PROGRAM ITMotion
VAR
	odometrie 			:FB_Motion_Odometrie;
END_VAR
VAR_INPUT
	IbPower				:BOOL;
	IbStop				:BOOL;
	IbPause				:BOOL;
	IbReset				:BOOL;
END_VAR
VAR_OUTPUT
	QbMoteurOn		:BOOL;
	QbMouvementTermine 	:BOOL;
END_VAR
VAR // added by the converter: edge detectors and wires of the graphical bodies
    _w1, _w2, _w3, _w4 : BOOL;
END_VAR

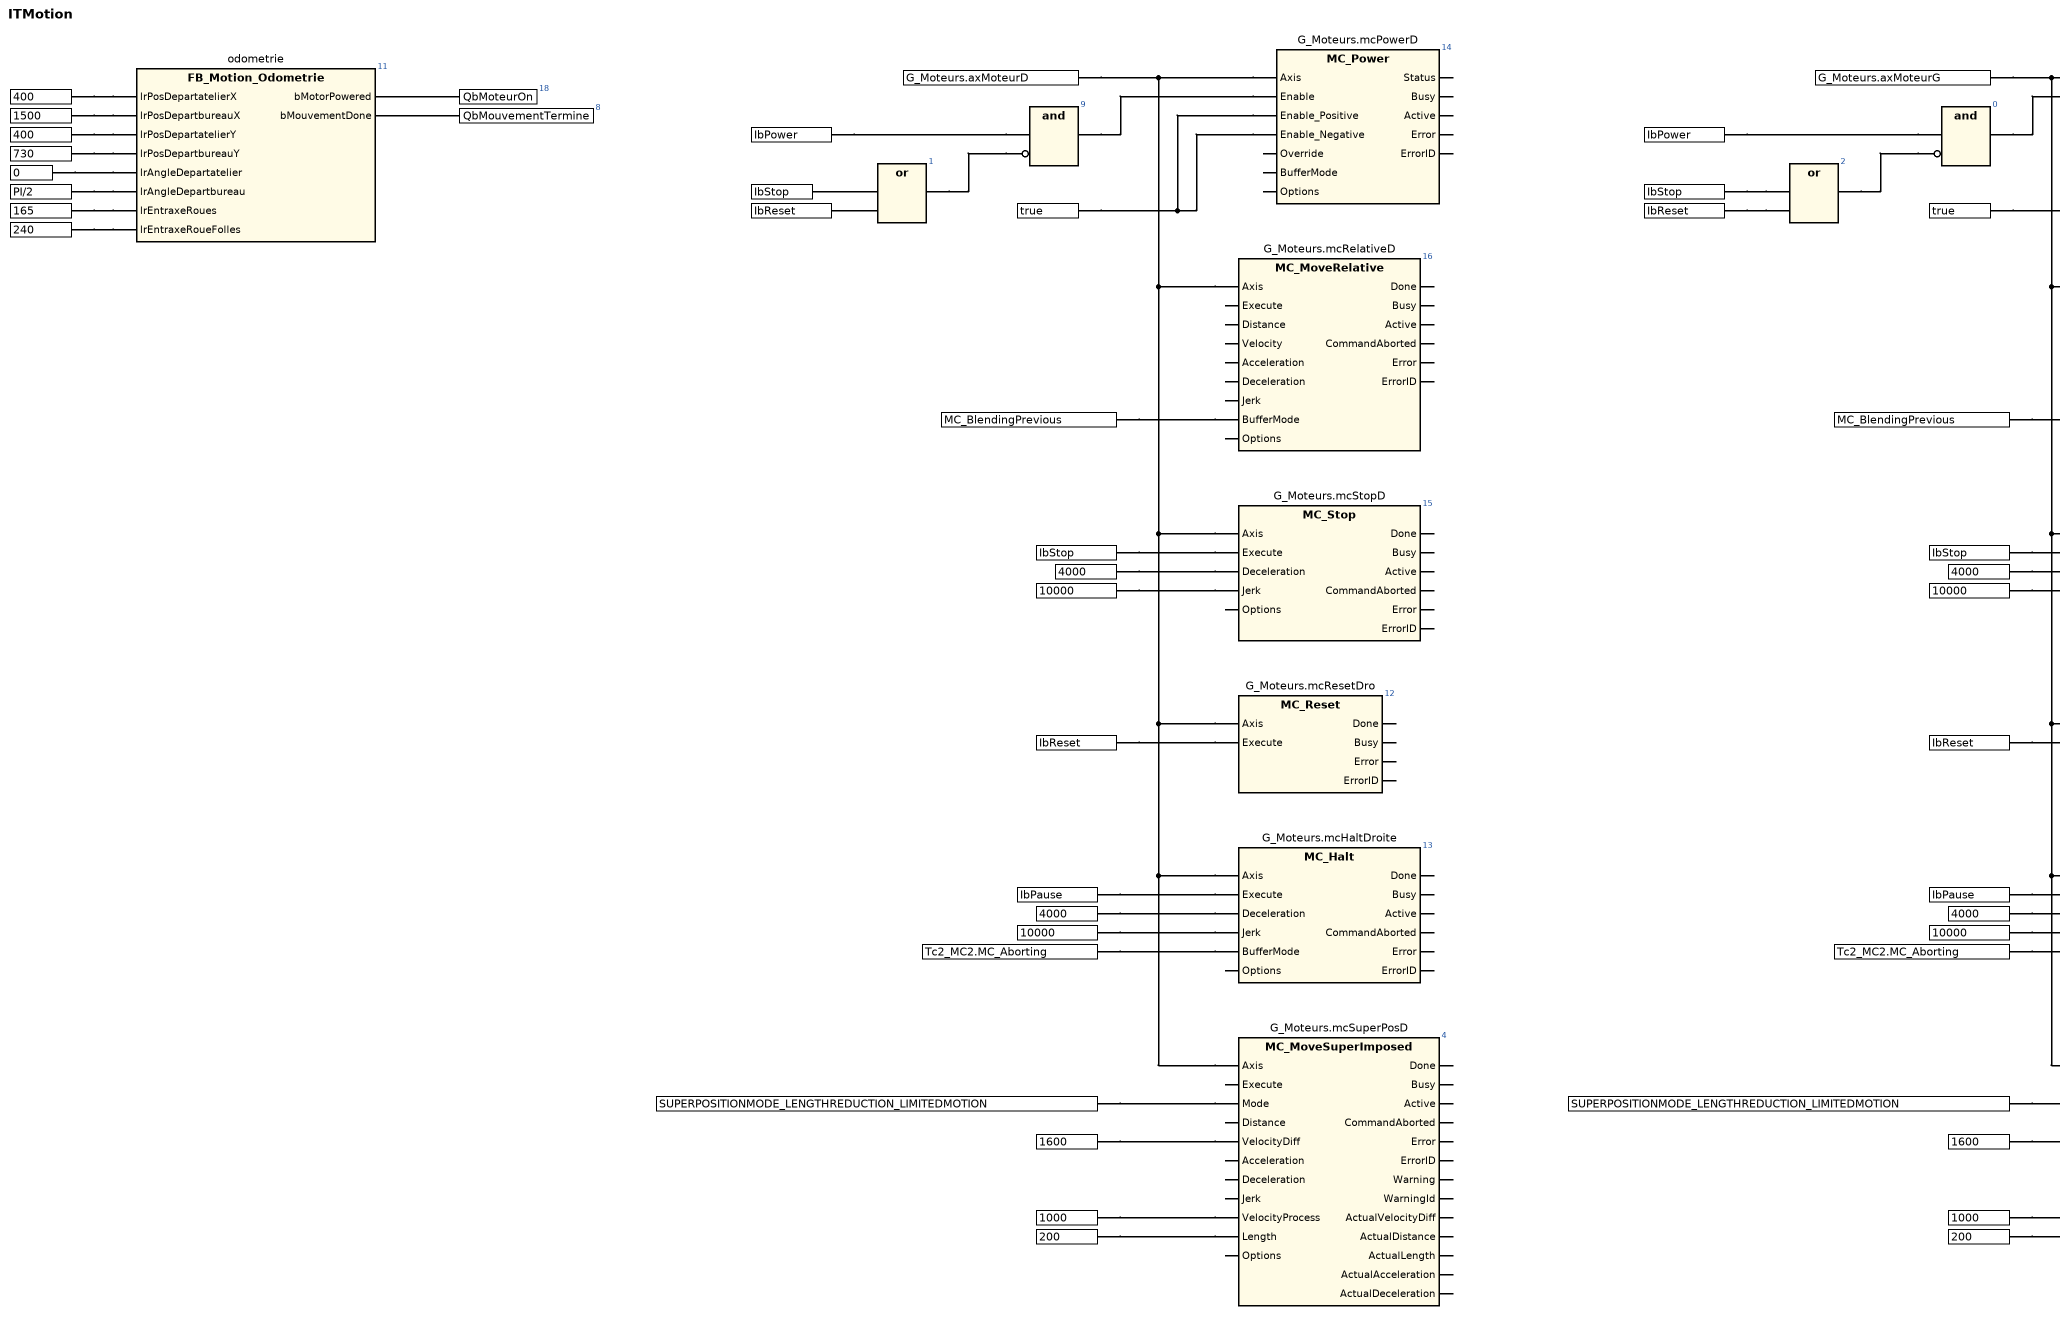
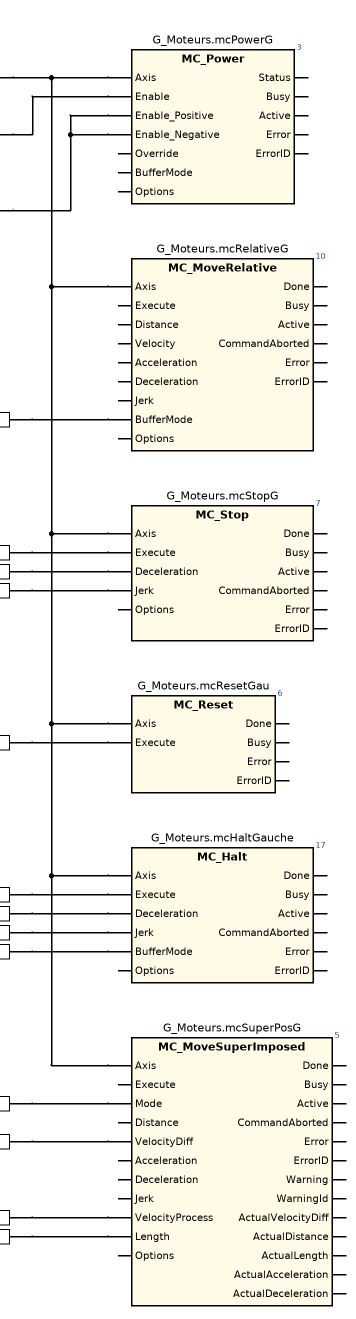
_w2 := IbPower AND NOT _w1;
_w3 := IbStop OR IbReset;
_w1 := IbStop OR IbReset;
G_Moteurs.mcPowerG(
    Axis := G_Moteurs.axMoteurG,
    Enable := _w2,
    Enable_Positive := true,
    Enable_Negative := true); // MC_Power
G_Moteurs.mcSuperPosD(
    Axis := G_Moteurs.axMoteurD,
    Mode := SUPERPOSITIONMODE_LENGTHREDUCTION_LIMITEDMOTION,
    VelocityDiff := 1600,
    VelocityProcess := 1000,
    Length := 200); // MC_MoveSuperImposed
G_Moteurs.mcSuperPosG(
    Axis := G_Moteurs.axMoteurG,
    Mode := SUPERPOSITIONMODE_LENGTHREDUCTION_LIMITEDMOTION,
    VelocityDiff := 1600,
    VelocityProcess := 1000,
    Length := 200); // MC_MoveSuperImposed
G_Moteurs.mcResetGau(Axis := G_Moteurs.axMoteurG, Execute := IbReset); // MC_Reset
G_Moteurs.mcStopG(Axis := G_Moteurs.axMoteurG, Execute := IbStop, Deceleration := 4000, Jerk := 10000); // MC_Stop
QbMouvementTermine := odometrie.bMouvementDone;
_w4 := IbPower AND NOT _w3;
G_Moteurs.mcRelativeG(Axis := G_Moteurs.axMoteurG, BufferMode := MC_BlendingPrevious); // MC_MoveRelative
odometrie(
    lrPosDepartatelierX := 400,
    lrPosDepartbureauX := 1500,
    lrPosDepartatelierY := 400,
    lrPosDepartbureauY := 730,
    lrAngleDepartatelier := 0,
    lrAngleDepartbureau := PI/2,
    lrEntraxeRoues := 165,
    lrEntraxeRoueFolles := 240); // FB_Motion_Odometrie
G_Moteurs.mcResetDro(Axis := G_Moteurs.axMoteurD, Execute := IbReset); // MC_Reset
G_Moteurs.mcHaltDroite(
    Axis := G_Moteurs.axMoteurD,
    Execute := IbPause,
    Deceleration := 4000,
    Jerk := 10000,
    BufferMode := Tc2_MC2.MC_Aborting); // MC_Halt
G_Moteurs.mcPowerD(
    Axis := G_Moteurs.axMoteurD,
    Enable := _w4,
    Enable_Positive := true,
    Enable_Negative := true); // MC_Power
G_Moteurs.mcStopD(Axis := G_Moteurs.axMoteurD, Execute := IbStop, Deceleration := 4000, Jerk := 10000); // MC_Stop
G_Moteurs.mcRelativeD(Axis := G_Moteurs.axMoteurD, BufferMode := MC_BlendingPrevious); // MC_MoveRelative
G_Moteurs.mcHaltGauche(
    Axis := G_Moteurs.axMoteurG,
    Execute := IbPause,
    Deceleration := 4000,
    Jerk := 10000,
    BufferMode := Tc2_MC2.MC_Aborting); // MC_Halt
QbMoteurOn := odometrie.bMotorPowered;

END_PROGRAM

(* stored: Version 1.1.0.1, ProductVersion 3.1.4024.12
   POU ITMotion: Id {fd64bfcf-93a1-4e1b-8879-06832046600a}, SpecialFunc None *)
